{attribute addProperty BoxType "AT2041-0250-0019"}
{attribute addProperty Id "A_0103_AT2042_5250_0018_AT2042_5250AT2042_C5E5984862678.25"}
{attribute addProperty CRC "1169792368"}
{attribute addProperty SizeInBites "626"}
{attribute addProperty SizeInBytes "78.25"}
TYPE A_0041_AT2041_0250_0019_45B99D70 EXTENDS AT2041_BA5A9548 :
STRUCT
	{attribute addProperty Name "A_0103_AT2042_5250_0018_AT2042_5250"}
	A_0103_AT2042_5250_0018_AT2042_5250 : AT2042_C5E59848;
END_STRUCT
END_TYPE

(* stored: Version 1.2.0.0, ProductVersion 3.1.4024.9
   DUT A_0041_AT2041_0250_0019_45B99D70: Id {c6675d98-3a03-43ef-a81d-8479f7594e94} *)
